FUNCTION_BLOCK Hutschienenmoped_XL_1_LED_strip (* Service Interface Function Block Type *)
  (* Function: All Inputs; Description: Copyright (c) 2018, 2023 Jose Cabral, HR Agrartechnik GmbH This program and the accompanying materials are made available under the terms of the Eclipse Public License 2.0 which is available at https://www.eclipse.org/legal/epl-2.0/ SPDX-License-Identifier: EPL-2.0 this maps to QX uses LED_GPIO_MODE *)
  (* Version 1.0, 2018-12-05, Jose Cabral *)
  (* Version 1.1, 2022-08-04, Franz Höpfinger, HR Agrartechnik GmbH *)
  (* Version 1.2, 2023-01-05, Franz Höpfinger, HR Agrartechnik GmbH *)
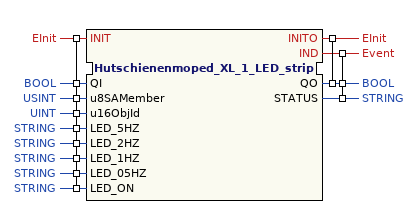
  EVENT_INPUT
    INIT : EInit WITH QI, u8SAMember, u16ObjId, LED_5HZ, LED_2HZ, LED_1HZ, LED_05HZ, LED_ON; (* Service Initialization *)
  END_EVENT
  EVENT_OUTPUT
    INITO : EInit WITH QO; (* Initialization Confirm *)
    IND WITH QO, STATUS; (* Indication from Resource *)
  END_EVENT
  VAR_INPUT
    QI : BOOL; (* Event Input Qualifier *)
    u8SAMember : USINT := Output_strip; (* Identify the Output Number of Strip *)
    u16ObjId : UINT := LED_GREEN; (* This identify the Colour. *)
    LED_5HZ : STRING; (* Identifier for LED blinking 5HZ, highest Prio (Prio 6) *)
    LED_2HZ : STRING; (* Identifier for LED blinking 2HZ, Prio 5 *)
    LED_1HZ : STRING; (* Identifier for LED blinking 1HZ, Prio 4 *)
    LED_05HZ : STRING; (* Identifier for LED blinking 0.5Hz, Prio 3 *)
    LED_ON : STRING; (* Identifier for LED always on, Prio 1 *)
  END_VAR
  VAR_OUTPUT
    QO : BOOL; (* Event Output Qualifier *)
    STATUS : STRING; (* Service Status *)
  END_VAR
END_FUNCTION_BLOCK
